(*

## Short summary
This class implements the interface `I32BitTimeAssertions`. 
It contains the assert statements for the data type ``TIME``

.. <legal notes>

legal notes
=================
| SPDX-FileCopyrightText: © 2022 ekvip automation GmbH <info@ekvip.de>
| SPDX-License-Identifier: Apache-2.0
| For details check: Apache-2.0_

.. _Apache-2.0: https://www.apache.org/licenses/LICENSE-2.0

.. </legal notes>

==

*)

{attribute 'reflection'}
FUNCTION_BLOCK INTERNAL SimpleTimeAssertions EXTENDS AbstractAssertion IMPLEMENTS I32BitTimeAssertions
VAR CONSTANT
	(* maximum value for the data type ``TIME`` *)
	MAX_TIME	:TIME := TO_TIME(16#FF_FF_FF_FF);
END_VAR

(*

## Short summary
This abstract property returns the class name of the concrete object, 
It's for debugging purpose

.. <legal notes>

legal notes
=================
| SPDX-FileCopyrightText: © 2022 ekvip automation GmbH <info@ekvip.de>
| SPDX-License-Identifier: Apache-2.0
| For details check: Apache-2.0_

.. _Apache-2.0: https://www.apache.org/licenses/LICENSE-2.0

.. </legal notes>

*)

PROPERTY className :CNM_AbstractObject.ClassName
GET
className := 'CNM_Assertor.SimplyTimeAssertions';
END_GET
END_PROPERTY

(*

## Short summary
This method returns the passed time since the timestamp was created

.. <legal notes>

legal notes
=================
| SPDX-FileCopyrightText: © 2022 ekvip automation GmbH <info@ekvip.de>
| SPDX-License-Identifier: Apache-2.0
| For details check: Apache-2.0_

.. _Apache-2.0: https://www.apache.org/licenses/LICENSE-2.0

.. </legal notes>


:return: passed time since ``startTime``

*)

METHOD PROTECTED getTimePassed :TIME
VAR_INPUT
	(* timestamp start *)
	startTime	:TIME;
END_VAR
VAR
	(* current time to calculate the passed time *)
	currentTime	:TIME;
END_VAR
currentTime := TIME();
IF (currentTime > startTime) THEN
	getTimePassed := (currentTime - startTime);
ELSE
	getTimePassed := ((THIS^.MAX_TIME - startTime) + currentTime);
END_IF
END_METHOD

(*

## Short summary
This assertion method checks whether time has elapsed since the timestamp time

.. <legal notes>

legal notes
=================
| SPDX-FileCopyrightText: © 2022 ekvip automation GmbH <info@ekvip.de>
| SPDX-License-Identifier: Apache-2.0
| For details check: Apache-2.0_

.. _Apache-2.0: https://www.apache.org/licenses/LICENSE-2.0

.. </legal notes>



*)

METHOD timeHasExpired
VAR_INPUT
	(* start time you get it with ``TIME()`` *)
	timestamp		:TIME;
	(* timeout like ``t#300ms`` *)
	expiringTime	:TIME;
	(* message if the assertion is false *)
	message			:AssertMessage;
END_VAR
VAR
	(* measured passed time *)
	passedTime		:TIME;
END_VAR
passedTime := THIS^.getTimePassed(timestamp);
IF (passedTime < expiringTime) THEN
	THIS^.assertionWasWrong(
		message			:= message,
		additionalText	:= THIS^.getDebugInfo('timeHasExpired')
	);	
END_IF
END_METHOD

(*

## Short summary
This assertion method checks that the time since the timestamp time has not yet elapsed

.. <legal notes>

legal notes
=================
| SPDX-FileCopyrightText: © 2022 ekvip automation GmbH <info@ekvip.de>
| SPDX-License-Identifier: Apache-2.0
| For details check: Apache-2.0_

.. _Apache-2.0: https://www.apache.org/licenses/LICENSE-2.0

.. </legal notes>



*)

METHOD timeHasNotExpired
VAR_INPUT
	(* start time you get it with ``TIME()`` *)
	timestamp		:TIME;
	(* timeout like ``t#300ms`` *)
	expiringTime	:TIME;
	(* message if the assertion is false *)
	message			:AssertMessage;
END_VAR
VAR
	(* measured passed time *)
	passedTime		:TIME;
END_VAR
passedTime := THIS^.getTimePassed(timestamp);
IF (passedTime >= expiringTime) THEN
	THIS^.assertionWasWrong(
		message			:= message,
		additionalText	:= THIS^.getDebugInfo('timeHasNotExpired')
	);	
END_IF
END_METHOD

(*

## Short summary
This assertion method checks if the current value is equal to the expected value

.. <legal notes>

legal notes
=================
| SPDX-FileCopyrightText: © 2022 ekvip automation GmbH <info@ekvip.de>
| SPDX-License-Identifier: Apache-2.0
| For details check: Apache-2.0_

.. _Apache-2.0: https://www.apache.org/licenses/LICENSE-2.0

.. </legal notes>



*)

METHOD valueIsEqualTo
VAR_INPUT
	(* current value to check *)
	currentValue	:TIME;
	(* expected value to compare *)
	expectedValue	:TIME;
	(* message if the assertion is false *)
	message			:AssertMessage;
END_VAR
IF (currentValue <> expectedValue) THEN
	THIS^.assertionWasWrong(
		message			:= message,
		additionalText	:= THIS^.getDebugInfo('valueIsEqualTo')
	);	
END_IF
END_METHOD

(*

## Short summary
This assertion method checks if the current value is greater than the less value

.. <legal notes>

legal notes
=================
| SPDX-FileCopyrightText: © 2022 ekvip automation GmbH <info@ekvip.de>
| SPDX-License-Identifier: Apache-2.0
| For details check: Apache-2.0_

.. _Apache-2.0: https://www.apache.org/licenses/LICENSE-2.0

.. </legal notes>



*)

METHOD valueIsGreaterThan
VAR_INPUT
	(* current value to check *)
	currentValue	:TIME;
	(* less than lower limit *)
	lessValue		:TIME;
	(* message if the assertion is false *)
	message			:AssertMessage;
END_VAR
IF (currentValue <= lessValue) THEN
	THIS^.assertionWasWrong(
		message			:= message,
		additionalText	:= THIS^.getDebugInfo('valueIsGreaterThan')
	);	
END_IF
END_METHOD

(*

## Short summary
This assertion method checks if the current value is inside a limit

**Attention:** 
	limits are included: ``valueIsInRangeOf(t#3ms,t#3ms ,t#3ms)`` is a true assertion

.. <legal notes>

legal notes
=================
| SPDX-FileCopyrightText: © 2022 ekvip automation GmbH <info@ekvip.de>
| SPDX-License-Identifier: Apache-2.0
| For details check: Apache-2.0_

.. _Apache-2.0: https://www.apache.org/licenses/LICENSE-2.0

.. </legal notes>



*)

METHOD valueIsInRangeOf
VAR_INPUT
	(* lower limit for the current value *)
	lowerLimit		:TIME;
	(* current value to check *)
	currentValue	:TIME;
	(* upper limit for the current value *)
	upperLimit		:TIME;
	(* message if the assertion is false *)
	message			:AssertMessage;
END_VAR
IF ((currentValue < lowerLimit) OR (currentValue > upperLimit)) THEN
	THIS^.assertionWasWrong(
		message			:= message,
		additionalText	:= THIS^.getDebugInfo('valueIsInRangeOf')
	);	
END_IF
END_METHOD

(*

## Short summary
This assertion method checks if the current value is less than the greater value

.. <legal notes>

legal notes
=================
| SPDX-FileCopyrightText: © 2022 ekvip automation GmbH <info@ekvip.de>
| SPDX-License-Identifier: Apache-2.0
| For details check: Apache-2.0_

.. _Apache-2.0: https://www.apache.org/licenses/LICENSE-2.0

.. </legal notes>



*)

METHOD valueIsLessThan
VAR_INPUT
	(* current value to check *)
	currentValue	:TIME;
	(* greater than upper limit *)
	greaterValue	:TIME;
	(* message if the assertion is false *)
	message			:AssertMessage;
END_VAR
IF (currentValue >= greaterValue) THEN
	THIS^.assertionWasWrong(
		message			:= message,
		additionalText	:= THIS^.getDebugInfo('valueIsLessThan')
	);	
END_IF
END_METHOD

(*

## Short summary
This assertion method checks if the current value is less than or equal to the maximum value

.. <legal notes>

legal notes
=================
| SPDX-FileCopyrightText: © 2022 ekvip automation GmbH <info@ekvip.de>
| SPDX-License-Identifier: Apache-2.0
| For details check: Apache-2.0_

.. _Apache-2.0: https://www.apache.org/licenses/LICENSE-2.0

.. </legal notes>



*)

METHOD valueIsMax
VAR_INPUT
	(* current value to check *)
	currentValue	:TIME;
	(* upper limit for the current value *)
	maximumValue	:TIME;
	(* message if the assertion is false *)
	message			:AssertMessage;
END_VAR
IF (currentValue > maximumValue) THEN
	THIS^.assertionWasWrong(
		message			:= message,
		additionalText	:= THIS^.getDebugInfo('valueIsMax')
	);	
END_IF
END_METHOD

(*

## Short summary
This assertion method checks if the current value is greater than or equal to the minimum value

.. <legal notes>

legal notes
=================
| SPDX-FileCopyrightText: © 2022 ekvip automation GmbH <info@ekvip.de>
| SPDX-License-Identifier: Apache-2.0
| For details check: Apache-2.0_

.. _Apache-2.0: https://www.apache.org/licenses/LICENSE-2.0

.. </legal notes>



*)

METHOD valueIsMin
VAR_INPUT
	(* current value to check *)
	currentValue	:TIME;
	(* lower limit for the current value *)
	minimumValue	:TIME;
	(* message if the assertion is false *)
	message			:AssertMessage;
END_VAR
IF (currentValue < minimumValue) THEN
	THIS^.assertionWasWrong(
		message			:= message,
		additionalText	:= THIS^.getDebugInfo('valueIsMin')
	);	
END_IF
END_METHOD

(*

## Short summary
This assertion method checks if the current value is not equal to the unexpected value

.. <legal notes>

legal notes
=================
| SPDX-FileCopyrightText: © 2022 ekvip automation GmbH <info@ekvip.de>
| SPDX-License-Identifier: Apache-2.0
| For details check: Apache-2.0_

.. _Apache-2.0: https://www.apache.org/licenses/LICENSE-2.0

.. </legal notes>



*)

METHOD valueIsNotEqualTo
VAR_INPUT
	(* current value to check *)
	currentValue	:TIME;
	(* unexpected value to compare *)
	unexpectedValue	:TIME;
	(* message if the assertion is false *)
	message			:AssertMessage;
END_VAR
IF (currentValue = unexpectedValue) THEN
	THIS^.assertionWasWrong(
		message			:= message,
		additionalText	:= THIS^.getDebugInfo('valueIsNotEqualTo')
	);	
END_IF
END_METHOD

END_FUNCTION_BLOCK

(* stored: Version 1.1.0.1, ProductVersion 3.1.4026.11
   POU SimpleTimeAssertions: Id {3dc4ef92-3bb4-4e95-b496-4aa32fc732a6}, SpecialFunc None
   Property className: Id {eab4cd17-0085-4f1f-8b00-1fc0a67f213f}
   Get Get: Id {545a483e-72e0-4cbc-8f12-93beafb0552a}
   Method getTimePassed: Id {b475e509-ce1a-4f36-bdf9-502b457f1cb3}
   Method timeHasExpired: Id {282aaaa0-e35f-4687-a261-2f78d8403978}
   Method timeHasNotExpired: Id {a18e6149-7689-45e6-a0c8-6095b98ddfdc}
   Method valueIsEqualTo: Id {2e5deb6d-1923-4f79-972d-c93b4d14a94f}
   Method valueIsGreaterThan: Id {def48364-b0ae-4795-b818-44199ea1782f}
   Method valueIsInRangeOf: Id {827cf796-573d-4dee-888a-37b4fcfe68fb}
   Method valueIsLessThan: Id {944426bc-aebf-4150-9ca9-8ad3a75b33e8}
   Method valueIsMax: Id {edb56a55-c256-471a-adc5-7e7580ef0587}
   Method valueIsMin: Id {61a6234f-68db-4573-b0cd-dae7ec5744e1}
   Method valueIsNotEqualTo: Id {c3386c38-bca0-41bf-a068-7c9a76e331dd} *)
